(* IEC 61131-3 sources: PLC_Defuser/Datasets/Water_tank/legitimate/lsubstitution_stop1, 1 file *)

(* ---- lsubstitution_stop1.st ---- *)
FUNCTION_BLOCK stop
  VAR_INPUT
    IN1 : BOOL;
  END_VAR
  VAR_OUTPUT
    OUT : BOOL;
  END_VAR

  IF IN1 = FALSE then
    OUT:=TRUE;
  else
    OUT:=FALSE;
  end_IF;
END_FUNCTION_BLOCK

FUNCTION_BLOCK valves_handler
  VAR_INPUT
    IN1 : INT;
    input1 : BOOL;
    IN_TLB1 : INT;
    IN_TLB2 : INT;
  END_VAR
  VAR_OUTPUT
    OUT_MV1 : BOOL;
    OUT_MV2 : BOOL;
  END_VAR
  VAR
    real_value : INT;
  END_VAR

  real_value :=  IN1 - 5;

  IF real_value <= IN_TLB2 then
    OUT_MV2 := FALSE;
    OUT_MV1 := TRUE;
  end_IF;

  IF real_value >= IN_TLB1 THEN
    OUT_MV2 := TRUE;
    OUT_MV1 := FALSE;
  end_IF;

  IF input1 = TRUE then
    OUT_MV2 := FALSE;
    OUT_MV1 := FALSE;
  end_IF;

END_FUNCTION_BLOCK

PROGRAM program0
  VAR_INPUT
    TLB2 : INT;
    TLB1 : INT;
    START : BOOL;
    input1 : BOOL;
    VALUE : INT;
  END_VAR
  VAR_OUTPUT
    MV1 : BOOL;
    MV2 : BOOL;
    CYCLE_ON : BOOL;
  END_VAR
  VAR
    stop0 : stop;
    valves_handler0 : valves_handler;
  END_VAR

  stop0(EN := CYCLE_ON OR START, IN1 := input1);
  CYCLE_ON := stop0.OUT;
  valves_handler0(EN := CYCLE_ON, IN1 := VALUE, input1 := input1, IN_TLB1 := TLB1, IN_TLB2 := TLB2);
  IF valves_handler0.ENO THEN
      MV1 := valves_handler0.OUT_MV1;
  END_IF;
  IF valves_handler0.ENO THEN
      MV2 := valves_handler0.OUT_MV2;
  END_IF;
END_PROGRAM

CONFIGURATION Config0

  RESOURCE Res0 ON PLC
    TASK task0(INTERVAL := T#20ms,PRIORITY := 0);
    PROGRAM instance0 WITH task0 : program0;
  END_RESOURCE
END_CONFIGURATION
